TYPE ST_Bel_RGBW_Zustand :
STRUCT
	Betrieb_Anford		: BOOL;
	Betrieb_Soll		: BOOL;
	Betrieb				: BOOL;

	Regelung_Modus		: SINT;

	Regelung_Istw		: REAL;
	Regelung_Sollw		: REAL;
	Steuerung_Istw		: REAL;
	Steuerung_Sollw		: REAL;


	Farbcode			: STRING;



	Leistung			: BYTE;	(* 0..100 % *)

	Freigabe			: BOOL;
	Freigabe_Deakt		: BOOL;
	Freigabe_Code		: WORD;
	Helligkeit			: REAL;
	Kommunikation		: BOOL;

	Lampen_Monitoring	: ARRAY [0..30] OF ST_Bel_Lampen_Monitoring;

	Stoerung				: BOOL;
	Stoerung_Code		: WORD;

	Warnung				: BOOL;
	Warnung_Code		: WORD;

	Status				: SINT;

	Status_Vorl			: BOOL;
	Status_Nachl			: BOOL;

	Quittierung			: BOOL;



END_STRUCT
END_TYPE

(* stored: Version 1.1.0.1, ProductVersion 3.1.4024.10
   DUT ST_Bel_RGBW_Zustand: Id {e93a5956-1d19-48c3-96ba-5c4bec599a91} *)
